Fanuc KAREL source: port_TPIN.kl

PROGRAM TP
%NOLOCKGROUP
VAR
 x: BOOLEAN
BEGIN
 x = TPIN[3]
END TP
